FUNCTION_BLOCK FB_HnhtHnltLinkage
VAR_INPUT
	//control struct for hnht hnlt linkage
	controlAutomatic : ST_HnhtHnltLinkageControl;
END_VAR
VAR_OUTPUT
END_VAR
VAR
	HeatExchanger1System : FB_HeatExchanger1System;
	
	//internal variables
	bAlgorithmPermission : BOOL;
END_VAR

bAlgorithmPermission := controlAutomatic.bAlgorithmPermission_HNHT AND controlAutomatic.bAlgorithmPermission_HNLT;

HeatExchanger1System(bSetStatusOnAutomatic := controlAutomatic.bSetStatusOn_HeatExchanger1,
	bAlgorithmPermission := bAlgorithmPermission,
	fSetPointAutomatic := controlAutomatic.fFeedTemperature_HNLT_Heating);

END_FUNCTION_BLOCK

(* stored: Version 1.1.0.1, ProductVersion 3.1.4024.10
   POU FB_HnhtHnltLinkage: Id {01f6a0de-a95a-4f6e-9757-ed042616c8fb}, SpecialFunc None *)
